# EPICS substitutions: BLDApp/Db/BLDMCastReceiverPcavs.substitutions
file BLDMCastReceiverPhaseCavity.template
{
#         Station			MC Group	Stat_Scan
pattern { STN			,	MC,			STAT_SCAN	}
        { "PhaseCavity"	,  	"1"			"5"	}
}
